// TIA Portal V19 export
FUNCTION_BLOCK "FC_Modbus_Arduino"   // FB1, LAD
{ S7_Optimized_Access := 'TRUE' }
// stored: MemoryReserve 100, SetENOAutomatically false
   VAR_INPUT
      Start_Feeder : Bool;
   END_VAR
   VAR_OUTPUT
      Feeder_Ready : Bool;
   END_VAR
BEGIN

REGION Network 1
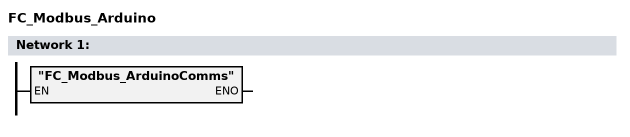
   RUNG wire#powerrail
      "FC_Modbus_ArduinoComms"()
   END_RUNG
   // the same network as SCL:
   "FC_Modbus_ArduinoComms"();
END_REGION
END_FUNCTION_BLOCK
